INTERFACE I_Vec4 EXTENDS I_Vec3


PROPERTY w : LREAL
GET
END_GET
END_PROPERTY

END_INTERFACE

(* stored: Version 1.1.0.1
   Itf I_Vec4: Id {d6831b85-2c4c-4d0a-b783-213a1dbe68b8}
   Property w: Id {1e2facaf-ec30-4cec-90d5-e084127bc0f9}
   Get Get: Id {8f4d5b69-a2e5-49ed-8aef-4c45ad79831d} *)
